FUNCTION Convert_LINT_TO_DINT : Hresult
VAR_INPUT
	in : LINT;
	out : REFERENCE TO DINT;
END_VAR
VAR
	converted : DINT;
END_VAR

converted := LINT_TO_DINT(in);

IF (DINT_TO_LINT(converted) <> in) THEN
	Convert_LINT_TO_DINT := INCOMPATIBLE;
	RETURN;
END_IF

out := converted;

END_FUNCTION

(* stored: Version 1.1.0.1, ProductVersion 3.1.4024.12
   POU Convert_LINT_TO_DINT: Id {948bcbfd-d14d-4a21-810a-24f245816c5c}, SpecialFunc None *)
